FUNCTION_BLOCK POU
VAR_INPUT
END_VAR
VAR_OUTPUT
END_VAR
VAR
END_VAR

STATECHART POU  // abortable
END_STATECHART

END_FUNCTION_BLOCK

(* stored: Version 1.1.0.1, ProductVersion 3.1.4024.3
   POU POU: Id {adee7f17-895a-4e47-a5e1-f2834cf7555d}, SpecialFunc None *)
